{attribute addProperty BoxType "EP1809-0042-0018"}
{attribute addProperty Id "DI_X01_Pin4AT %I*DI_X01_Pin_E4AEF59E810DI_X01_Pin2AT %I*DI_X01_Pin_E4AEF59E810DI_X02_Pin4AT %I*DI_X02_Pin_E4AEF59E810DI_X02_Pin2AT %I*DI_X02_Pin_E4AEF59E810DI_X03_Pin4AT %I*DI_X03_Pin_E4AEF59E810DI_X03_Pin2AT %I*DI_X03_Pin_E4AEF59E810DI_X04_Pin4AT %I*DI_X04_Pin_E4AEF59E810DI_X04_Pin2AT %I*DI_X04_Pin_E4AEF59E810DI_X05_Pin4AT %I*DI_X05_Pin_E4AEF59E810DI_X05_Pin2AT %I*DI_X05_Pin_E4AEF59E810DI_X06_Pin4AT %I*DI_X06_Pin_E4AEF59E810DI_X06_Pin2AT %I*DI_X06_Pin_E4AEF59E810DI_X07_Pin4AT %I*DI_X07_Pin_E4AEF59E810DI_X07_Pin2AT %I*DI_X07_Pin_E4AEF59E810DI_X08_Pin4AT %I*DI_X08_Pin_E4AEF59E810DI_X08_Pin2AT %I*DI_X08_Pin_E4AEF59E810WcStateAT %I*WcState_F855686C1620InfoDataAT %I*InfoData_192954DE1620"}
{attribute addProperty CRC "3134433351"}
{attribute addProperty SizeInBites "160"}
{attribute addProperty SizeInBytes "20"}
TYPE EP1809_FA80E4F8 :
STRUCT
	{attribute addProperty Name "DI_X01_Pin4"}
	DI_X01_Pin4 : DI_X01_Pin_E4AEF59E;
	{attribute addProperty Name "DI_X01_Pin2"}
	DI_X01_Pin2 : DI_X01_Pin_E4AEF59E;
	{attribute addProperty Name "DI_X02_Pin4"}
	DI_X02_Pin4 : DI_X02_Pin_E4AEF59E;
	{attribute addProperty Name "DI_X02_Pin2"}
	DI_X02_Pin2 : DI_X02_Pin_E4AEF59E;
	{attribute addProperty Name "DI_X03_Pin4"}
	DI_X03_Pin4 : DI_X03_Pin_E4AEF59E;
	{attribute addProperty Name "DI_X03_Pin2"}
	DI_X03_Pin2 : DI_X03_Pin_E4AEF59E;
	{attribute addProperty Name "DI_X04_Pin4"}
	DI_X04_Pin4 : DI_X04_Pin_E4AEF59E;
	{attribute addProperty Name "DI_X04_Pin2"}
	DI_X04_Pin2 : DI_X04_Pin_E4AEF59E;
	{attribute addProperty Name "DI_X05_Pin4"}
	DI_X05_Pin4 : DI_X05_Pin_E4AEF59E;
	{attribute addProperty Name "DI_X05_Pin2"}
	DI_X05_Pin2 : DI_X05_Pin_E4AEF59E;
	{attribute addProperty Name "DI_X06_Pin4"}
	DI_X06_Pin4 : DI_X06_Pin_E4AEF59E;
	{attribute addProperty Name "DI_X06_Pin2"}
	DI_X06_Pin2 : DI_X06_Pin_E4AEF59E;
	{attribute addProperty Name "DI_X07_Pin4"}
	DI_X07_Pin4 : DI_X07_Pin_E4AEF59E;
	{attribute addProperty Name "DI_X07_Pin2"}
	DI_X07_Pin2 : DI_X07_Pin_E4AEF59E;
	{attribute addProperty Name "DI_X08_Pin4"}
	DI_X08_Pin4 : DI_X08_Pin_E4AEF59E;
	{attribute addProperty Name "DI_X08_Pin2"}
	DI_X08_Pin2 : DI_X08_Pin_E4AEF59E;
	{attribute addProperty Name "WcState"}
	WcState : WcState_F855686C;
	{attribute addProperty Name "InfoData"}
	InfoData : InfoData_192954DE;
END_STRUCT
END_TYPE

(* stored: Version 1.2.0.0, ProductVersion 3.1.4024.9
   DUT EP1809_FA80E4F8: Id {e8e46c80-f4df-4d62-a813-4d730e66b109} *)
